// TIA Portal V17 export
// export: Created 2024-09-03T21:54:46.8290554Z, ExportSetting WithDefaults, DisplayName Totally Integrated Automation Portal, DisplayVersion V17 Update 7, DisplayName TIA Portal Openness, DisplayVersion V17 Update 7, DisplayName TIA Portal Version Control Interface, DisplayVersion V17, DisplayName SINAMICS Startdrive Advanced, DisplayVersion V17 SP2, DisplayName SINAMICS Startdrive G110M, G120, G120C, G120D, G120P, G115D, DisplayVersion V17 SP2, DisplayName SINAMICS Startdrive G130, G150, S120, S150, SINAMICS MV, S210, DisplayVersion V17 SP2, DisplayName STEP 7 Professional, DisplayVersion V17 Update 7, DisplayName STEP 7 Safety, DisplayVersion V17 Update 6, DisplayName WinCC Advanced / Unified PC, DisplayVersion V17 Update 7
FUNCTION_BLOCK "RobotJob"   // FB45, GRAPH
VERSION : 0.1
// stored: AcknowledgeErrorsRequired true, AutoNumber true, GraphVersion 6.0, InitialValuesAcquisition false, IsIECCheckEnabled false, LanguageInNetworks LAD, LockOperatingMode false, PermanentILProcessingInMANMode false, SetENOAutomatically false, SkipSteps false, UDAEnableTagReadback false, WithAlarmHandling true
   // inherited from GRAPH_BASE
   VAR
      OFF_SQ_BASE : Bool;
   END_VAR
   VAR_INPUT
      OFF_SQ { ExternalAccessible := 'False'; ExternalVisible := 'False'; ExternalWritable := 'False'} : Bool := false;   // Turn sequence off
      INIT_SQ { ExternalAccessible := 'False'; ExternalVisible := 'False'; ExternalWritable := 'False'} : Bool := false;   // Set sequence to initial state
      ACK_EF { ExternalAccessible := 'False'; ExternalVisible := 'False'; ExternalWritable := 'False'} : Bool := false;   // Acknowledge all errors and faults
      S_PREV { ExternalAccessible := 'False'; ExternalVisible := 'False'; ExternalWritable := 'False'} : Bool := false;   // Output previous step in parameter S_NO
      S_NEXT { ExternalAccessible := 'False'; ExternalVisible := 'False'; ExternalWritable := 'False'} : Bool := false;   // Indicate next step in parameter S_NO
      SW_AUTO { ExternalAccessible := 'False'; ExternalVisible := 'False'; ExternalWritable := 'False'} : Bool := false;   // Automatic mode
      SW_TAP { ExternalAccessible := 'False'; ExternalVisible := 'False'; ExternalWritable := 'False'} : Bool := false;   // Semiautomatic/switch with transition
      SW_TOP { ExternalAccessible := 'False'; ExternalVisible := 'False'; ExternalWritable := 'False'} : Bool := false;   // Semiautomatic/ignore transition
      SW_MAN { ExternalAccessible := 'False'; ExternalVisible := 'False'; ExternalWritable := 'False'} : Bool := false;   // Manual mode
      S_SEL { ExternalAccessible := 'False'; ExternalVisible := 'False'; ExternalWritable := 'False'} : Int := 0;   // Select step to be output to S_NO
      S_ON { ExternalAccessible := 'False'; ExternalVisible := 'False'; ExternalWritable := 'False'} : Bool := false;   // Activate step indicated in S_NO
      S_OFF { ExternalAccessible := 'False'; ExternalVisible := 'False'; ExternalWritable := 'False'} : Bool := false;   // Deactivate step indicated S_NO
      T_PUSH { ExternalAccessible := 'False'; ExternalVisible := 'False'; ExternalWritable := 'False'} : Bool := false;   // Enable transition to switch in semi automatic mode
   END_VAR
   VAR_OUTPUT
      S_NO { ExternalAccessible := 'False'; ExternalVisible := 'False'; ExternalWritable := 'False'} : Int := 0;   // Step number
      S_MORE { ExternalAccessible := 'False'; ExternalVisible := 'False'; ExternalWritable := 'False'} : Bool := false;   // More steps are available and can be shown in S_NO
      S_ACTIVE { ExternalAccessible := 'False'; ExternalVisible := 'False'; ExternalWritable := 'False'} : Bool := false;   // Step indicated in S_NO is active
      ERR_FLT { ExternalAccessible := 'False'; ExternalVisible := 'False'; ExternalWritable := 'False'} : Bool := false;   // Interlock or supervision group error
      AUTO_ON { ExternalAccessible := 'False'; ExternalVisible := 'False'; ExternalWritable := 'False'} : Bool := false;   // Automatic mode is active
      TAP_ON { ExternalAccessible := 'False'; ExternalVisible := 'False'; ExternalWritable := 'False'} : Bool := false;   // Semiautomatic mode/step with transition enabled
      TOP_ON { ExternalAccessible := 'False'; ExternalVisible := 'False'; ExternalWritable := 'False'} : Bool := false;   // Semiautomatic mode/ignore transition enabled
      MAN_ON { ExternalAccessible := 'False'; ExternalVisible := 'False'; ExternalWritable := 'False'} : Bool := false;   // Manual mode is active
   END_VAR
BEGIN
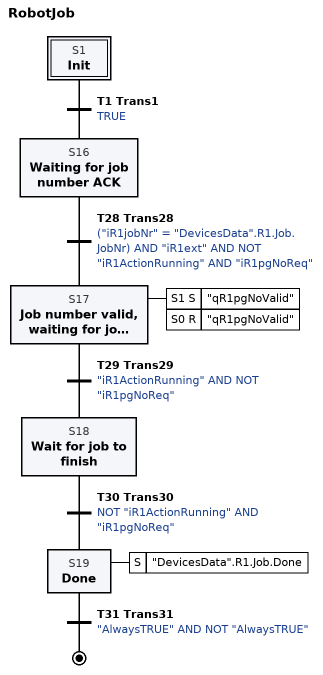
   // permanent pre-instructions
   NETWORK 1
      "DevicesData".R1.Job.Done := FALSE;

   // sequencer 1
   INITIAL_STEP Init:   // S1, max time T#10S, warning time T#7S
   END_STEP
   TRANSITION Trans1 FROM Init TO "Waiting for job number ACK"   // T1
      := TRUE;
   END_TRANSITION
   STEP "Waiting for job number ACK":   // S16, max time T#10S, warning time T#7S
      supervision V := #"Waiting for job number ACK".T > #"Waiting for job number ACK".T_MAX;
   END_STEP
   TRANSITION Trans28 FROM "Waiting for job number ACK" TO "Job number valid, waiting for job start"   // T28
      := ("iR1jobNr" = "DevicesData".R1.Job.JobNr) AND "iR1ext" AND NOT "iR1ActionRunning" AND "iR1pgNoReq";
   END_TRANSITION
   STEP "Job number valid, waiting for job start":   // S17, max time T#10S, warning time T#7S
      supervision V := #"Job number valid, waiting for job start".T > #"Job number valid, waiting for job start".T_MAX;
          S1  S    "qR1pgNoValid"
          S0  R    "qR1pgNoValid"
   END_STEP
   TRANSITION Trans29 FROM "Job number valid, waiting for job start" TO "Wait for job to finish"   // T29
      := "iR1ActionRunning" AND NOT "iR1pgNoReq";
   END_TRANSITION
   STEP "Wait for job to finish":   // S18, max time T#30S, warning time T#7S
      supervision V := #"Wait for job to finish".T > #"Wait for job to finish".T_MAX;
   END_STEP
   TRANSITION Trans30 FROM "Wait for job to finish" TO Done   // T30
      := NOT "iR1ActionRunning" AND "iR1pgNoReq";
   END_TRANSITION
   STEP Done:   // S19, max time T#10S, warning time T#7S
              S    "DevicesData".R1.Job.Done
   END_STEP
   TRANSITION Trans31 FROM Done TO END   // T31
      := "AlwaysTRUE" AND NOT "AlwaysTRUE";
   END_TRANSITION
END_FUNCTION_BLOCK
